// Mitsubishi GX Works2 project: Teoreti2   PLC: FX3G

// global labels: Global1
VAR_GLOBAL
  Wash_Machine AT Y001 : BOOL;
  Pressure_130 AT X002 : BOOL;
  Sensor_130 AT X002 : BOOL;
  Sensor_200 AT X003 : BOOL;
  Y5t AT Y005 : BOOL;
  Min_Z AT Y010 : BOOL;
END_VAR
VAR_GLOBAL CONSTANT
  Count10Cars : INT := 10;
END_VAR
VAR_GLOBAL
  Counter10Cars AT CS1 : BOOL;
  Fill_Soap AT Y004 : BOOL;
  Min_Soap AT Y011 : BOOL;
END_VAR

// task Task_01 (event TRUE, interval 0, priority 31): POU_01

PROGRAM POU_01
(* structured ladder/FBD written out as ST: instructions are called as NAME(EN, inputs, outputs); _pN, _eN, _tN stand for wires *)
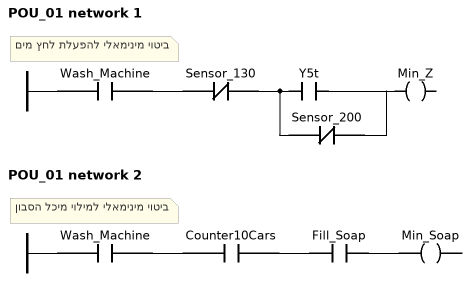
(* network 1 *)
(* ביטוי מינימאלי להפעלת לחץ מים *)
_p1 := Wash_Machine AND NOT Sensor_130;
Min_Z := (_p1 AND Y5t) OR (_p1 AND NOT Sensor_200);
(* network 2 *)
(* ביטוי מינימאלי למילוי מיכל הסבון *)
Min_Soap := Wash_Machine AND Counter10Cars AND Fill_Soap;
END_PROGRAM
